DATA_BLOCK "DB_End_MLZ_PLT"
TITLE =%version: 0.04 % CN: 20
//History:
//This version  %created_by:  nlhdl %
//              %date_created:  Tuesday, September 06, 2016 8:35:08 AM %
//              %release: VI_RAW/RA_Dev %
//
//Modification History:                                   By:    Date:     Rev:
//----------------------------------------------------  -------  --------  -----
//ra#16917: Update the MLZ according MCFV decomposition nlHdL    06-09-16   0.04
//ra#16917: Update the MLZ according MCFV decomposition nlHdL    06-09-16   0.04
//7324: ECS-P General from the RD to RA for platform    nlHdL    06-07-15   0.04
//15797: Keyword release added                          nlwwij   26-09-13   0.04
//14506: Add Motor_Stopped to EQP Basic & Lean          nlHdL    02-09-13   0.03
//CR19512 Update sources according S7 Manager           nlHdL    07-03-13   0.02
//Initial revision                                      nlcsu    21-12-11   0.01
//
FAMILY : RAW
VERSION : 0.0


  STRUCT
   Entries_Used : INT ;	//Number of entries used in tracking DB
   Displacement : INT ;	//Displacement last PLC cycle used by read tracking functions
   Entries_Present : INT ;	//Number of entries present in tracking DB
   DB_PLT_nr_Upstream : INT ;	//DB PLT number of the upstream
   DB_PLT_nr_Downstream : INT ;	//DB PLT number of the downstream
   Done : BOOL ;	//Header data is written in the PLT DB.
   Section_Run : BOOL ;	//Section running signal
   Motor_On_Speed : BOOL ;	//Motor on speed signal
   Cascade_Start_up : BOOL ;	//Cascade start up downstream
   Section_Available : BOOL ;	//Section is available to recieve items (TEP=1)
   Section_Operational : BOOL ;	//Section is started
   Item_at_Handover : BOOL ;	//Item at Handover position
   PEC_Latch : BOOL ;	//PEC Latch at EOS
   Inhibit_Receive_Item : BOOL ;	//Section is setting the inhibit to receive item found in upstream handover
   Section_Stopped : BOOL ;	//Section is stopped. (Actuele speed = 0)
   Length_Section : INT ;	//Length of the conveyor
   Entry : ARRAY  [1 .. 20 ] OF STRUCT
    Position : INT ;
    Info_State : WORD ;	//W#1x PEC, W#2x Owner, W#x4 Claimed, W#x8 Virtual, PEC W#x1 /2 /3, Owner W#3x /4
    Info_Physical : INT ;	//1= Leading Edge, 2= Trailing Edge, -3= Energy Save
    Link : INT ;
   END_STRUCT ;
  END_STRUCT ;
BEGIN
END_DATA_BLOCK

